RoboDK station: codealpha_task2.rdk

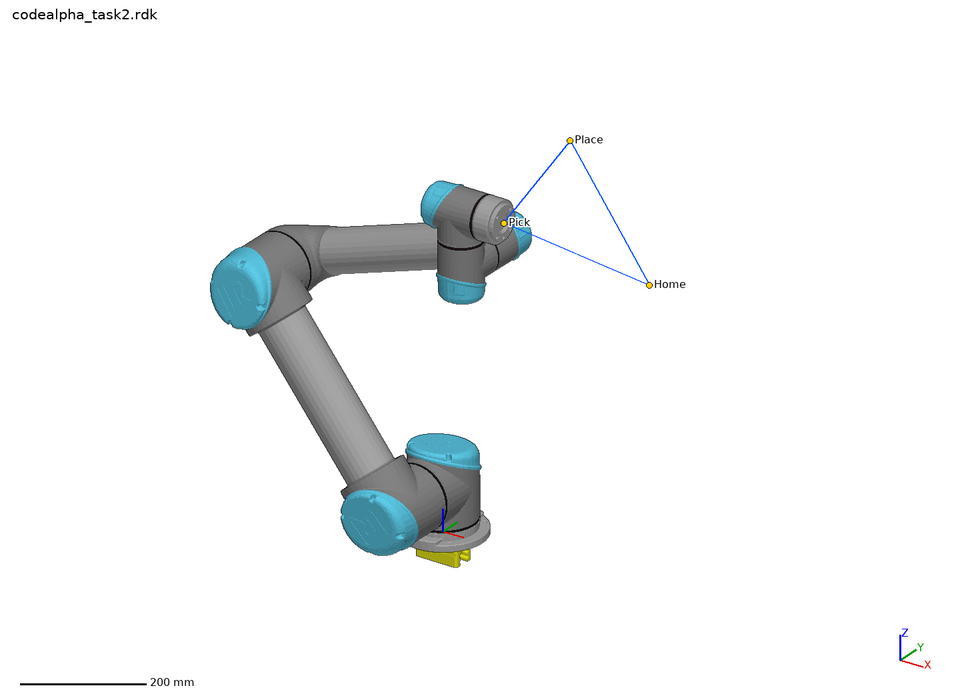
[picture v0: the station drawn from its stored meshes, robots at their saved joint values, targets as dots, program paths as lines]
Station New Station (1) (saved by RoboDK 6.0.4). Poses are relative to the parent item; angles as X-Y-Z fixed-axis rotations.
  - frame UR5 Base at (0, 1000, 0) mm
    - robot UR5: 6 axes
        modified DH rows (alpha deg, a mm, theta deg, d mm): 0, 0, 0, 89.2; 90, 0, 180, 0; 0, 425, 0, 0; 0, 392, 0, 109.3; -90, 0, 0, 94.75; 90, 0, 180, 82.5
        joint limits [-360, -360, -360, -360, -360, -360] to [360, 360, 360, 360, 360, 360]; home [0, -90, -90, 0, 90, 0]; saved at [0, -52, -110, -18, 90, 0]
    - robot Gripper: 1 axes
        joint limits [-40] to [0]; home [0]; saved at [0]
      - tool O-ring, TCP at (0, 0, 200) mm, size 37 x 37 x 3 mm, geometry from O-ring.stl
    - target Home (Cartesian target) at (474.5, -109.3, 608.95) mm, rotated rx -90 ry 0 rz -90 deg; joints [0, -90, -90, 0, 90, 0] of UR5
    - target Pick (Cartesian target) at (193.66, -109.3, 639.99) mm, rotated rx -90 ry 0 rz -90 deg; joints [0, -52, -110, -18, 90, 0] of UR5
    - target Place (Cartesian target) at (109.3, 193.66, 639.99) mm, rotated rx -90 ry 0 rz 0 deg; joints [90, -52, -110, -18, 90, 0] of UR5
  - program Prog1 (7 instructions, listed below)
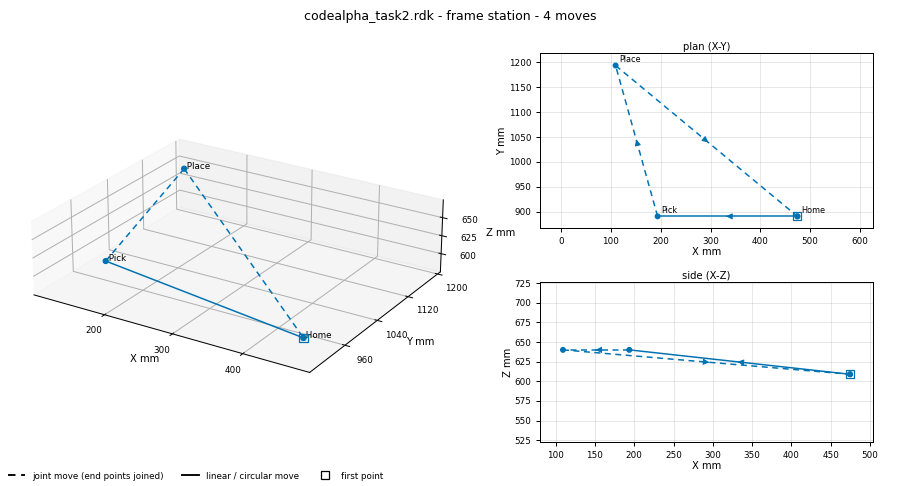
[picture p0: tool path of codealpha_task2.rdk in frame station, 4 of 4 moves have a stored position in this frame; points joined in program order, loops and branches not executed]

--- program Prog1 (robot UR5) ---
  Set Ref.: UR5 Base
  MoveJ (Home)
  MoveL (Pick)
  Attach to O-ring
  MoveJ (Place)
  Detach from O-ring
  MoveJ (Home)
